FUNCTION_BLOCK FB_PI_Controller
VAR_INPUT
	Reset				: BOOL; // Reset integral component
	ProcessVariable 	: LREAL;
	Setpoint			: LREAL;
	Kp					: LREAL;
	IntegralConstant 	: LREAL; // Repeats per minute
	RepeatsPerMinute	: BOOL := TRUE; // if false, repeats per second.
	MaxLoopOutput		: LREAL;
	MinLoopOutput		: LREAL;
	Bias				: LREAL;
END_VAR
VAR_OUTPUT
	Output 	: LREAL;
END_VAR
VAR
	p 		: FB_P_Control;
	i 		: FB_I_Controller;
	preClampedOutput : LREAL;
END_VAR

p(
	ProcessVariable:= ProcessVariable, 
	Setpoint:= Setpoint, 
	Kp:= Kp 
);

i(
	ProcessVariable := ProcessVariable, 
	Setpoint := Setpoint, 
	Ki	:= IntegralConstant / SEL(RepeatsPerMinute, 1, 60) , // normalising to repeats per minute. FB_I_COntroller block works in repeats per second natively.
	Pause := (preClampedOutput > MaxLoopOutput) OR (preClampedOutput < MinLoopOutput) ,
	Reset := Reset
);

// caclculate output
preClampedOutput := p.Term + i.Term + Bias;
Output := LIMIT( MinLoopOutput, preClampedOutput, MaxLoopOutput ); // clamp the output

END_FUNCTION_BLOCK

(* stored: Version 1.1.0.1, ProductVersion 3.1.4022.3
   POU FB_PI_Controller: Id {667c926c-65f6-42bc-9d46-ef9968266b60}, SpecialFunc None *)
